# EPICS substitutions: iocs/smartMotorIOC/iocBoot/iocSmartMotor/SmartMotor.substitutions
file "$(MOTOR)/db/motor.db"
{
pattern
{P,           N,      M,        DTYP,      C,  S,  DESC,          EGU,      DIR,  VELO,  VBAS,  ACCL,  BDST,  BVEL,  BACC,  MRES,  PREC,  DHLM,  DLLM,  INIT}
{smartMotor:, 1,  "m$(N)",  "SmartMotor",  0,  0,  "motor $(N)",  degrees,  Pos,  1,     .1,    .2,    0,     1,     .2,    0.01,  5,     100,   -100,  ""}
}
